// TIA Portal V17 export
FUNCTION "FC_FanGasControl" : Void   // FC, LAD
{ S7_Optimized_Access := 'TRUE' }
BEGIN

REGION Network 1: 风机输出
   // 风机运行按常开+风机故障反馈常闭→风机运行线圈；手动选择MOVE自动输出或MUL手动频率×2→控制输出
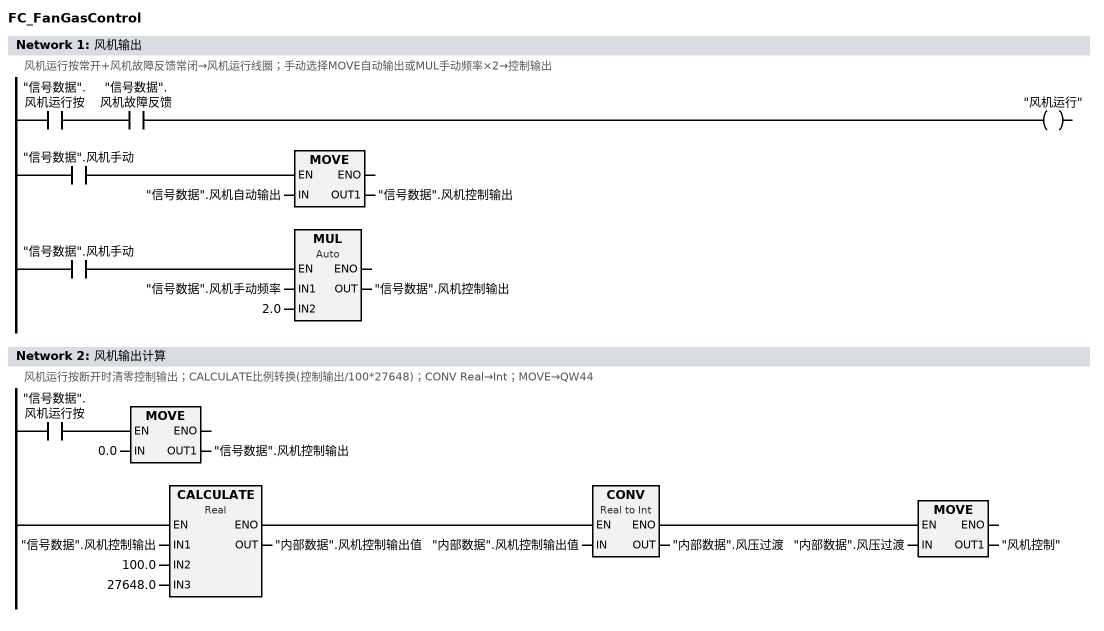
   RUNG wire#powerrail
      Contact( "信号数据".风机运行按 )
      Contact( "信号数据".风机故障反馈 )
      Coil( "风机运行" )
   END_RUNG
   RUNG wire#powerrail
      Contact( "信号数据".风机手动 )
      Move(in := "信号数据".风机自动输出, out1 => "信号数据".风机控制输出)
   END_RUNG
   RUNG wire#powerrail
      Contact( "信号数据".风机手动 )
      Mul(in1 := "信号数据".风机手动频率, in2 := 2.0, out => "信号数据".风机控制输出)
   END_RUNG
   // the same network as SCL:
   "风机运行" := "信号数据".风机运行按 AND "信号数据".风机故障反馈;
   IF "信号数据".风机手动 THEN
       "信号数据".风机控制输出 := "信号数据".风机自动输出;
       "信号数据".风机控制输出 := "信号数据".风机手动频率 * 2.0;
   END_IF;
END_REGION

REGION Network 2: 风机输出计算
   // 风机运行按断开时清零控制输出；CALCULATE比例转换(控制输出/100*27648)；CONV Real→Int；MOVE→QW44
   RUNG wire#powerrail
      Contact( "信号数据".风机运行按 )
      Move(in := 0.0, out1 => "信号数据".风机控制输出)
   END_RUNG
   RUNG wire#powerrail
      { S7_Templates := "SrcType := Real"; S7_Expression := "(IN1/IN2)*IN3" } Calculate(in1 := "信号数据".风机控制输出, in2 := 100.0, in3 := 27648.0, out => "内部数据".风机控制输出值)
      { S7_Templates := "[SrcType := Real, DestType := Int]" } Convert(in := "内部数据".风机控制输出值, out => "内部数据".风压过渡)
      Move(in := "内部数据".风压过渡, out1 => "风机控制")
   END_RUNG
   // the same network as SCL:
   IF "信号数据".风机运行按 THEN "信号数据".风机控制输出 := 0.0; END_IF;
   "内部数据".风机控制输出值 := ("信号数据".风机控制输出/100.0)*27648.0;
   "内部数据".风压过渡 := REAL_TO_INT("内部数据".风机控制输出值);
   "风机控制" := "内部数据".风压过渡;
END_REGION
END_FUNCTION
